(* Logix 5000 project; controller Sucrose_Main Emulate 5570 rev 20.12; software revision 20.01; part 9 of 30 *)
(* tags used below, declared in another part *)
   Alarm_ACK_Master_Timer : TIMER;
   DI_E20_0 : ALIAS FOR FLX_E20:0:I;   // Discrete Input EN2T_FLX 192.168.1.20
   DI_E20_1 : ALIAS FOR FLX_E20:1:I;   // Discrete Input EN2T_FLX 192.168.1.20
   DI_E20_2 : ALIAS FOR FLX_E20:2:I;   // Discrete Input EN2T_FLX 192.168.1.20
   DO_E20_3 : ALIAS FOR FLX_E20:3:O;   // Discrete Output EN2T_FLX 192.168.1.20
   DO_E20_4 : ALIAS FOR FLX_E20:4:O;   // Discrete Output EN2T_FLX 192.168.1.20
   DO_E20_5 : ALIAS FOR FLX_E20:5:O;   // Discrete Output EN2T_FLX 192.168.1.20
   FV230222_AOI : QSI_Flow_Valve;   // FV-23-02-22-O SUCROSE TANK #2 TO TRANSFER PUMP #2 MIX PROOF VALVE OPEN
   FV230412_AOI : QSI_Flow_Valve;   // FV-23-04-12-O SUCROSE TANK #2 TO TRANSFER PUMP #1 MIX PROOF VALVE OPEN
   FV230413_AOI : QSI_Flow_Valve;   // FV-23-04-13-O SUCROSE TANK #3 TO TRANSFER PUMP #1 MIX PROOF VALVE OPEN
   FV230421_AOI : QSI_Flow_Valve;   // FV-23-04-21-O SUCROSE TANK #1 TO TRANSFER PUMP #2 MIX PROOF VALVE OPEN
   FV230423_AOI : QSI_Flow_Valve;   // FV-23-04-23-O SUCROSE TANK #3 TO TRANSFER PUMP #2 MIX PROOF VALVE OPEN
   FV230441_AOI : QSI_Flow_Valve;   // FV-23-04-41-O SUCROSE TRANSFER PUMP #1 DISCHARGE TO FILTRATRION MIX PROOF VALVE OPEN
   FV230442_AOI : QSI_Flow_Valve;   // FV-23-04-42-O SUCROSE TRANSFER PUMP #2 DISCHARGE TO FILTRATRION MIX PROOF VALVE OPEN
   PBL1604001_AOI : QSI_Discrete_Device;   // PBL-16040-01 RESET PB LIGHT
   Sucrose_MM_Enable : BOOL;
   SucroseCIP_P230401_REMOTE : CIP_REMOTE;
   SucroseCIP_P230402_REMOTE : CIP_REMOTE;
   SucroseCIP_RINGMAIN_REMOTE : CIP_REMOTE;
   SucroseDischarge : Area_Program;
   SucroseFiltration : Area_Program;
   SucroseTanks : Area_Program;
(* DischargeArea_EN2T_IO_Discrete_DO_E20_3, continued *)

ROUTINE _03_FV230412   (* ladder *)
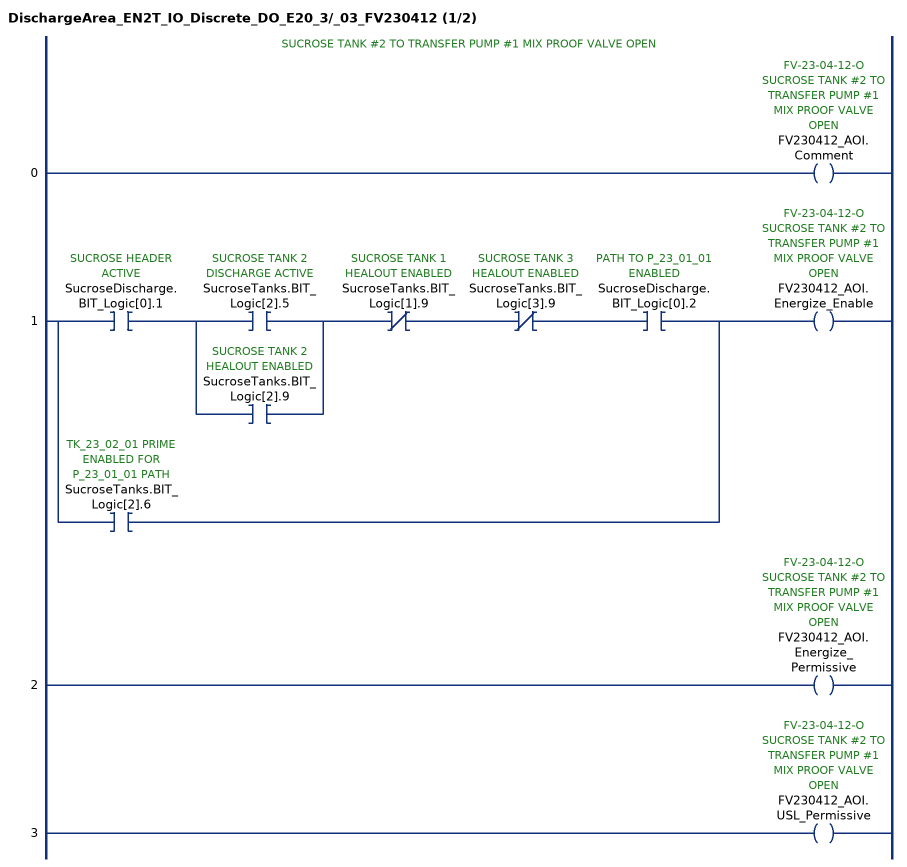
   // SUCROSE TANK #2 TO TRANSFER PUMP #1 MIX PROOF VALVE OPEN
   0: OTE(FV230412_AOI.Comment);
   1: [XIC(SucroseDischarge.BIT_Logic[0].1) [XIC(SucroseTanks.BIT_Logic[2].5) ,XIC(SucroseTanks.BIT_Logic[2].9) ] XIO(SucroseTanks.BIT_Logic[1].9) XIO(SucroseTanks.BIT_Logic[3].9) XIC(SucroseDischarge.BIT_Logic[0].2) ,XIC(SucroseTanks.BIT_Logic[2].6) ]OTE(FV230412_AOI.Energize_Enable);
   2: OTE(FV230412_AOI.Energize_Permissive);
   3: OTE(FV230412_AOI.USL_Permissive);
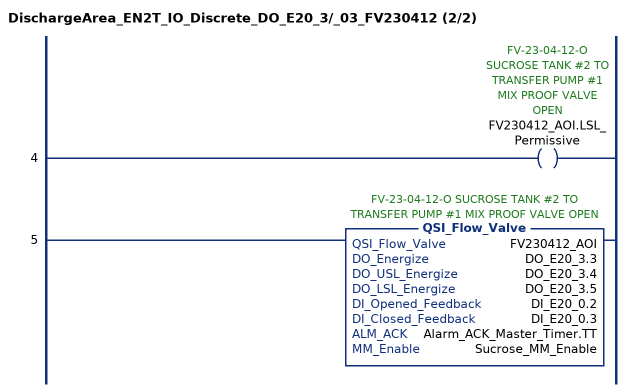
   4: OTE(FV230412_AOI.LSL_Permissive);
   5: QSI_Flow_Valve(FV230412_AOI,DO_E20_3.3,DO_E20_3.4,DO_E20_3.5,DI_E20_0.2,DI_E20_0.3,Alarm_ACK_Master_Timer.TT,Sucrose_MM_Enable);
END_ROUTINE

ROUTINE _06_FV230413   (* ladder *)
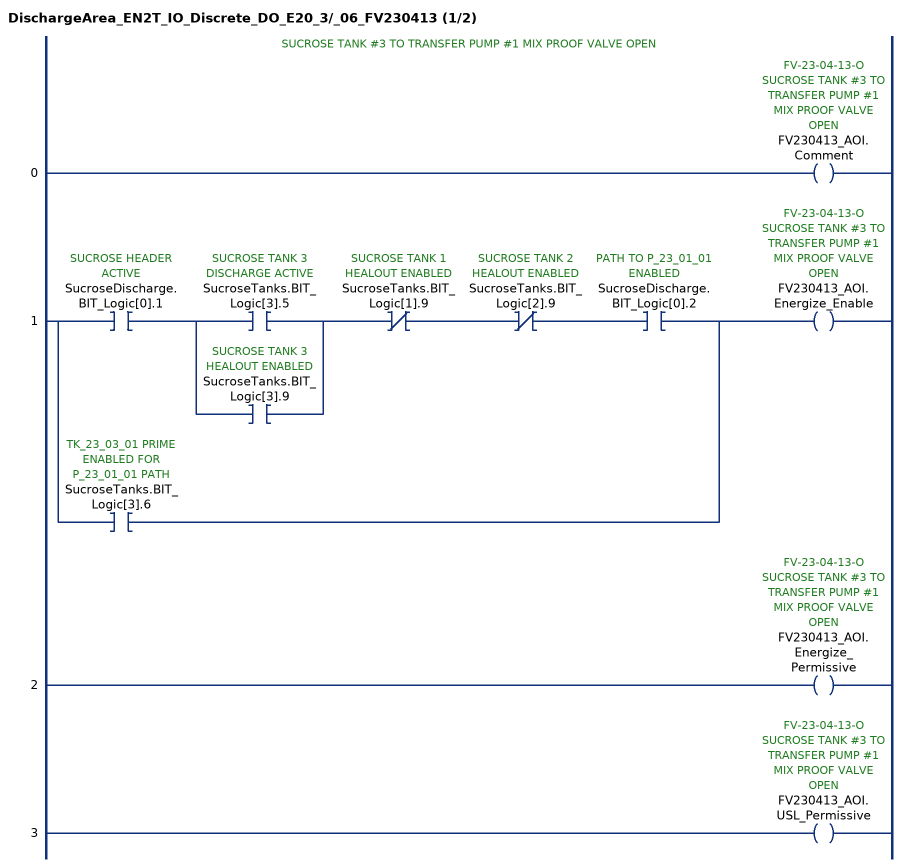
   // SUCROSE TANK #3 TO TRANSFER PUMP #1 MIX PROOF VALVE OPEN
   0: OTE(FV230413_AOI.Comment);
   1: [XIC(SucroseDischarge.BIT_Logic[0].1) [XIC(SucroseTanks.BIT_Logic[3].5) ,XIC(SucroseTanks.BIT_Logic[3].9) ] XIO(SucroseTanks.BIT_Logic[1].9) XIO(SucroseTanks.BIT_Logic[2].9) XIC(SucroseDischarge.BIT_Logic[0].2) ,XIC(SucroseTanks.BIT_Logic[3].6) ]OTE(FV230413_AOI.Energize_Enable);
   2: OTE(FV230413_AOI.Energize_Permissive);
   3: OTE(FV230413_AOI.USL_Permissive);
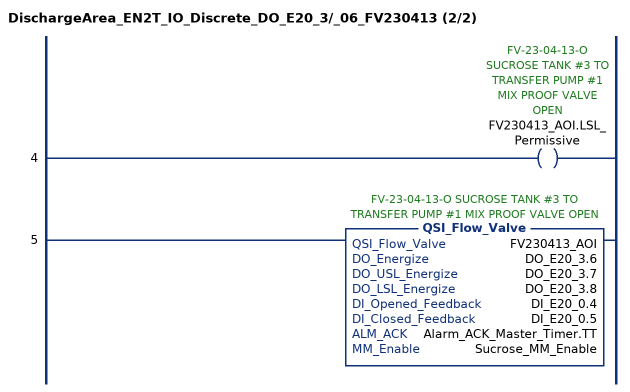
   4: OTE(FV230413_AOI.LSL_Permissive);
   5: QSI_Flow_Valve(FV230413_AOI,DO_E20_3.6,DO_E20_3.7,DO_E20_3.8,DI_E20_0.4,DI_E20_0.5,Alarm_ACK_Master_Timer.TT,Sucrose_MM_Enable);
END_ROUTINE

ROUTINE _09_FV230441   (* ladder *)
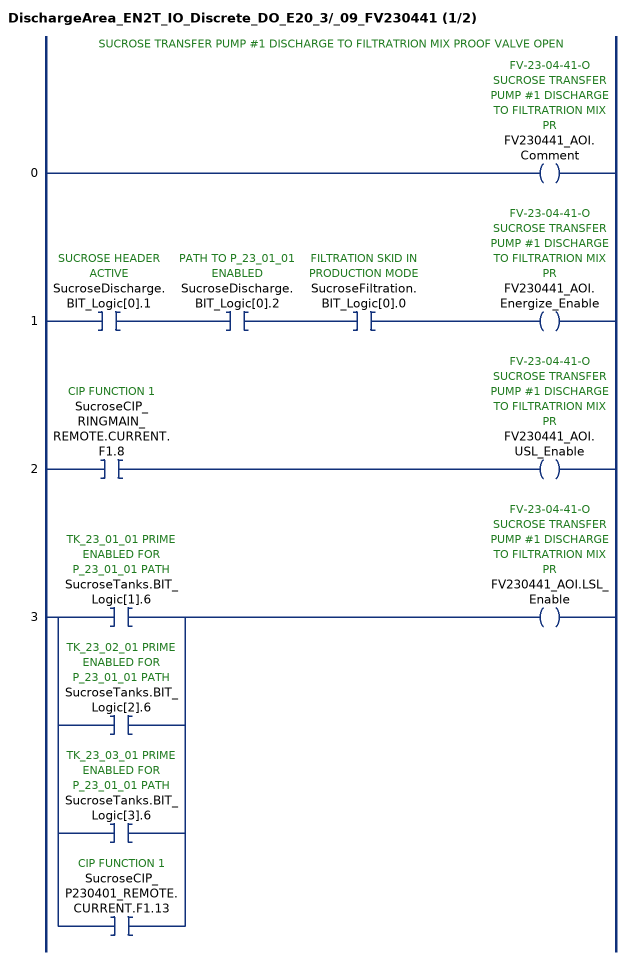
   // SUCROSE TRANSFER PUMP #1 DISCHARGE TO FILTRATRION MIX PROOF VALVE OPEN
   0: OTE(FV230441_AOI.Comment);
   1: XIC(SucroseDischarge.BIT_Logic[0].1)XIC(SucroseDischarge.BIT_Logic[0].2)XIC(SucroseFiltration.BIT_Logic[0].0)OTE(FV230441_AOI.Energize_Enable);
   2: XIC(SucroseCIP_RINGMAIN_REMOTE.CURRENT.F1.8)OTE(FV230441_AOI.USL_Enable);
   3: [XIC(SucroseTanks.BIT_Logic[1].6) ,XIC(SucroseTanks.BIT_Logic[2].6) ,XIC(SucroseTanks.BIT_Logic[3].6) ,XIC(SucroseCIP_P230401_REMOTE.CURRENT.F1.13) ]OTE(FV230441_AOI.LSL_Enable);
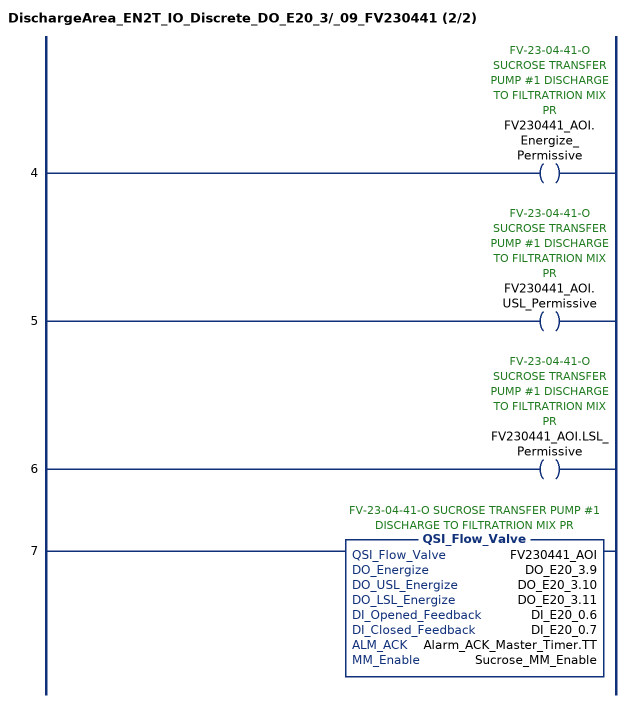
   4: OTE(FV230441_AOI.Energize_Permissive);
   5: OTE(FV230441_AOI.USL_Permissive);
   6: OTE(FV230441_AOI.LSL_Permissive);
   7: QSI_Flow_Valve(FV230441_AOI,DO_E20_3.9,DO_E20_3.10,DO_E20_3.11,DI_E20_0.6,DI_E20_0.7,Alarm_ACK_Master_Timer.TT,Sucrose_MM_Enable);
END_ROUTINE

ROUTINE _12_FV230442   (* ladder *)
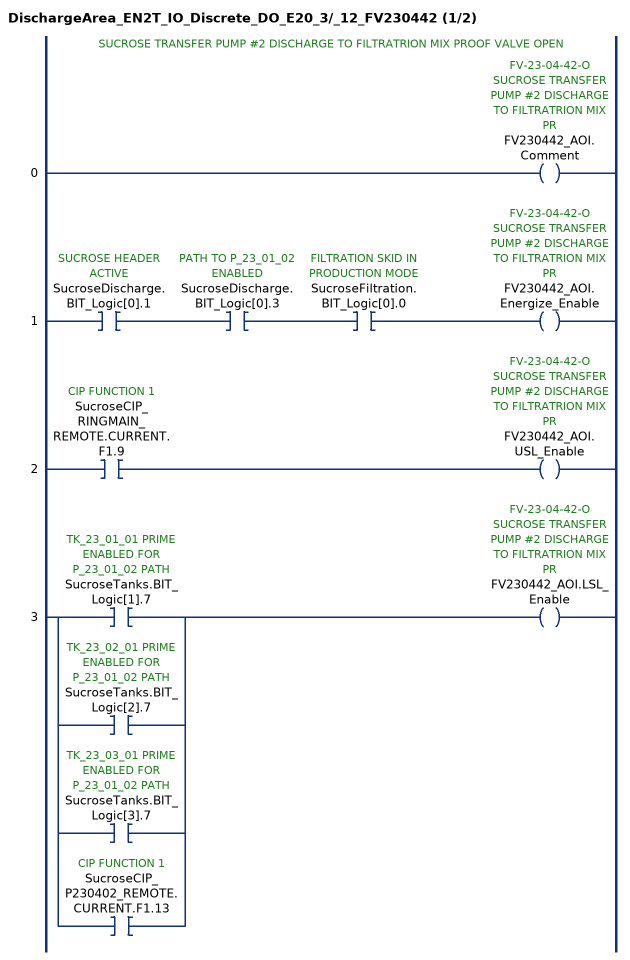
   // SUCROSE TRANSFER PUMP #2 DISCHARGE TO FILTRATRION MIX PROOF VALVE OPEN
   0: OTE(FV230442_AOI.Comment);
   1: XIC(SucroseDischarge.BIT_Logic[0].1)XIC(SucroseDischarge.BIT_Logic[0].3)XIC(SucroseFiltration.BIT_Logic[0].0)OTE(FV230442_AOI.Energize_Enable);
   2: XIC(SucroseCIP_RINGMAIN_REMOTE.CURRENT.F1.9)OTE(FV230442_AOI.USL_Enable);
   3: [XIC(SucroseTanks.BIT_Logic[1].7) ,XIC(SucroseTanks.BIT_Logic[2].7) ,XIC(SucroseTanks.BIT_Logic[3].7) ,XIC(SucroseCIP_P230402_REMOTE.CURRENT.F1.13) ]OTE(FV230442_AOI.LSL_Enable);
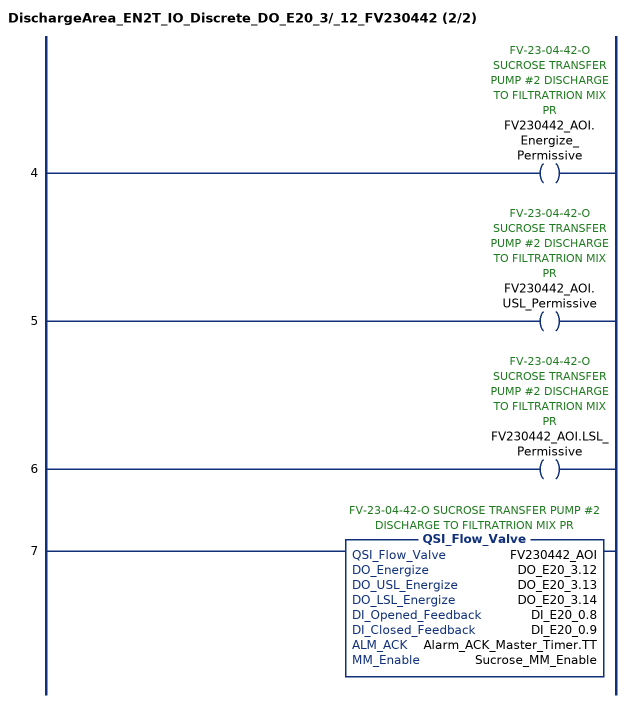
   4: OTE(FV230442_AOI.Energize_Permissive);
   5: OTE(FV230442_AOI.USL_Permissive);
   6: OTE(FV230442_AOI.LSL_Permissive);
   7: QSI_Flow_Valve(FV230442_AOI,DO_E20_3.12,DO_E20_3.13,DO_E20_3.14,DI_E20_0.8,DI_E20_0.9,Alarm_ACK_Master_Timer.TT,Sucrose_MM_Enable);
END_ROUTINE

ROUTINE MainRoutine   (* ladder *)
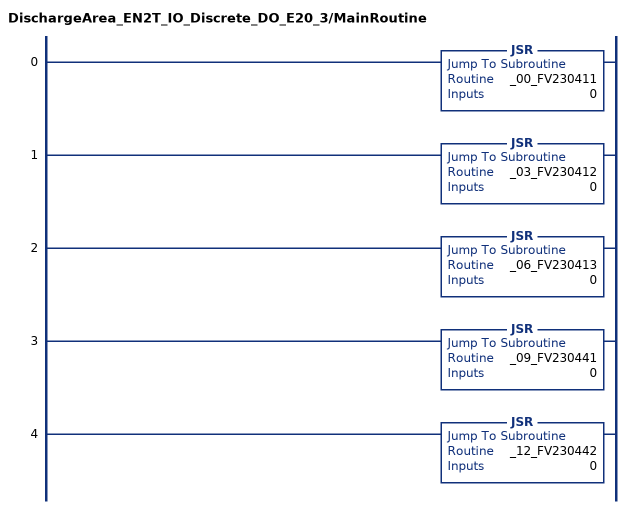
   0: JSR(_00_FV230411,0);
   1: JSR(_03_FV230412,0);
   2: JSR(_06_FV230413,0);
   3: JSR(_09_FV230441,0);
   4: JSR(_12_FV230442,0);
END_ROUTINE
END_PROGRAM

PROGRAM DischargeArea_EN2T_IO_Discrete_DO_E20_4   (* main routine MainRoutine *)

ROUTINE _03_FV230421   (* ladder *)
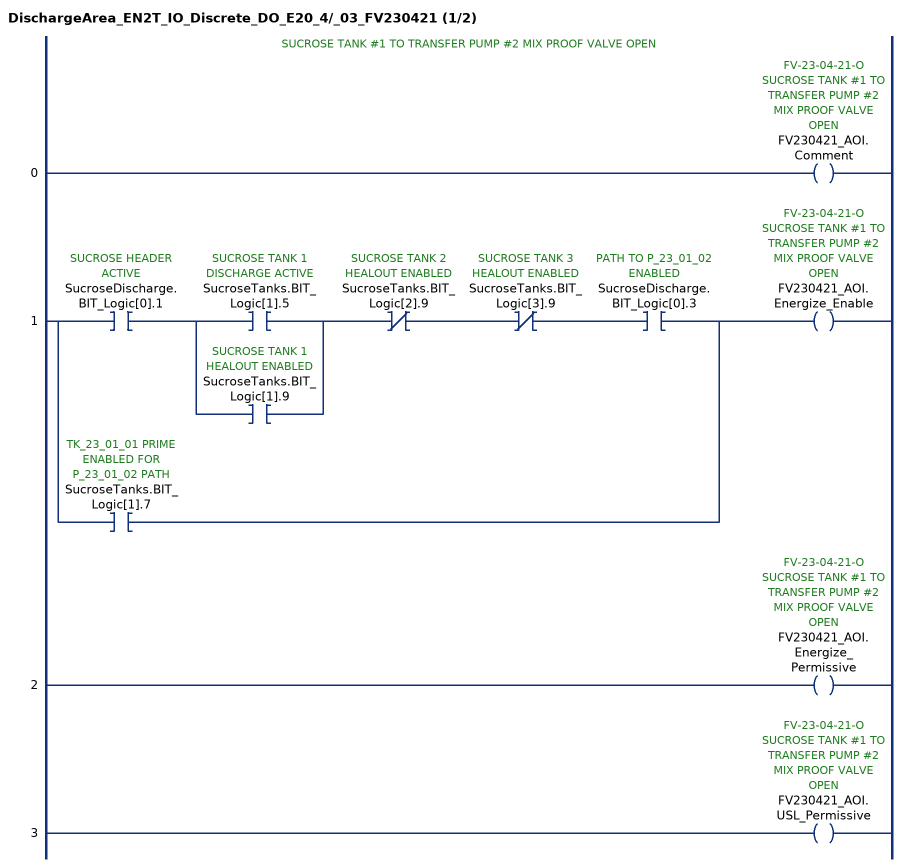
   // SUCROSE TANK #1 TO TRANSFER PUMP #2 MIX PROOF VALVE OPEN
   0: OTE(FV230421_AOI.Comment);
   1: [XIC(SucroseDischarge.BIT_Logic[0].1) [XIC(SucroseTanks.BIT_Logic[1].5) ,XIC(SucroseTanks.BIT_Logic[1].9) ] XIO(SucroseTanks.BIT_Logic[2].9) XIO(SucroseTanks.BIT_Logic[3].9) XIC(SucroseDischarge.BIT_Logic[0].3) ,XIC(SucroseTanks.BIT_Logic[1].7) ]OTE(FV230421_AOI.Energize_Enable);
   2: OTE(FV230421_AOI.Energize_Permissive);
   3: OTE(FV230421_AOI.USL_Permissive);
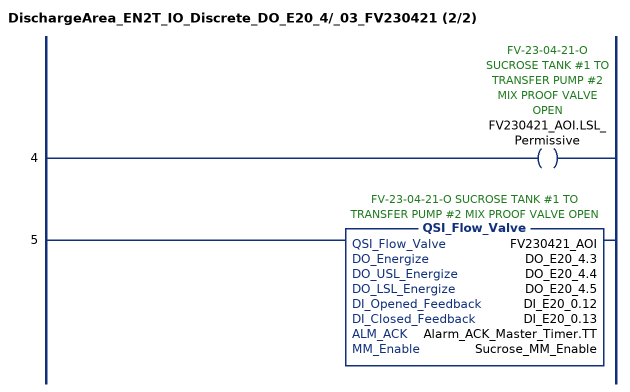
   4: OTE(FV230421_AOI.LSL_Permissive);
   5: QSI_Flow_Valve(FV230421_AOI,DO_E20_4.3,DO_E20_4.4,DO_E20_4.5,DI_E20_0.12,DI_E20_0.13,Alarm_ACK_Master_Timer.TT,Sucrose_MM_Enable);
END_ROUTINE

ROUTINE _06_FV230222   (* ladder *)
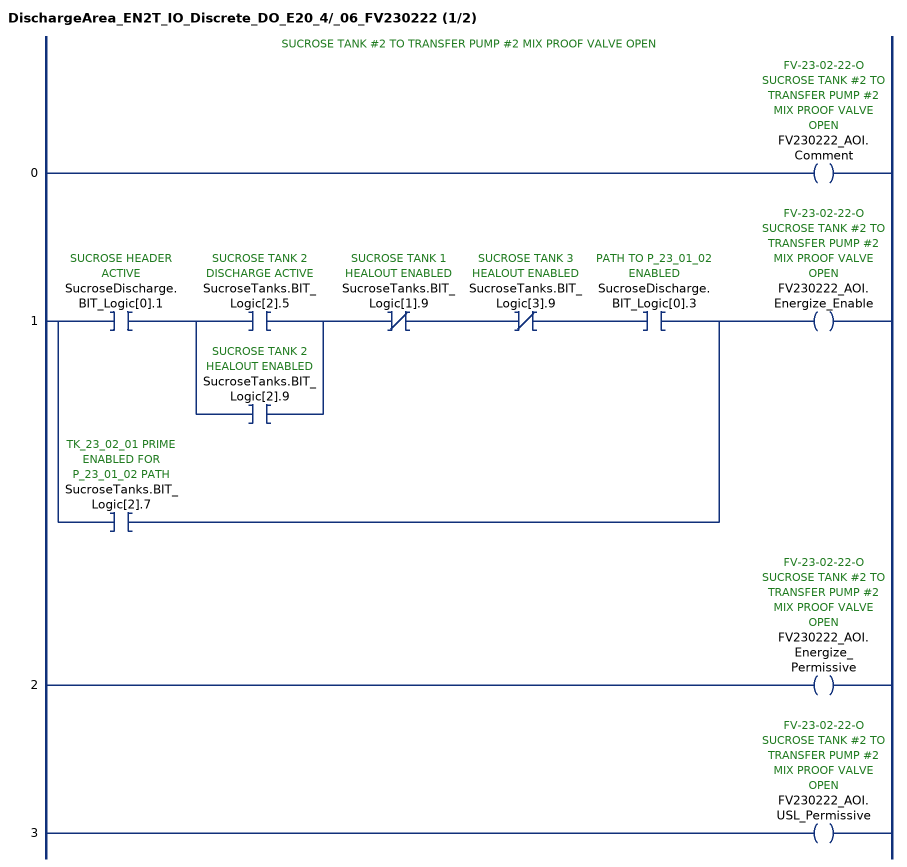
   // SUCROSE TANK #2 TO TRANSFER PUMP #2 MIX PROOF VALVE OPEN
   0: OTE(FV230222_AOI.Comment);
   1: [XIC(SucroseDischarge.BIT_Logic[0].1) [XIC(SucroseTanks.BIT_Logic[2].5) ,XIC(SucroseTanks.BIT_Logic[2].9) ] XIO(SucroseTanks.BIT_Logic[1].9) XIO(SucroseTanks.BIT_Logic[3].9) XIC(SucroseDischarge.BIT_Logic[0].3) ,XIC(SucroseTanks.BIT_Logic[2].7) ]OTE(FV230222_AOI.Energize_Enable);
   2: OTE(FV230222_AOI.Energize_Permissive);
   3: OTE(FV230222_AOI.USL_Permissive);
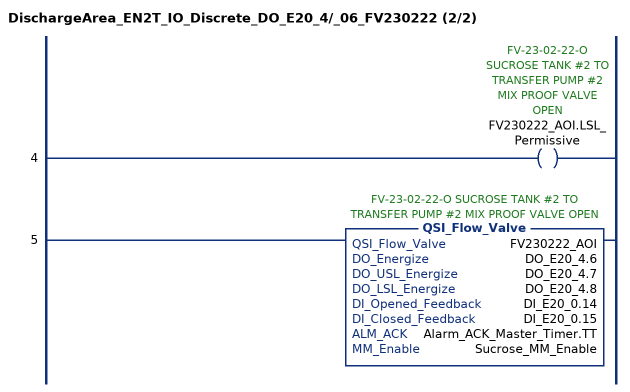
   4: OTE(FV230222_AOI.LSL_Permissive);
   5: QSI_Flow_Valve(FV230222_AOI,DO_E20_4.6,DO_E20_4.7,DO_E20_4.8,DI_E20_0.14,DI_E20_0.15,Alarm_ACK_Master_Timer.TT,Sucrose_MM_Enable);
END_ROUTINE

ROUTINE _09_FV230423   (* ladder *)
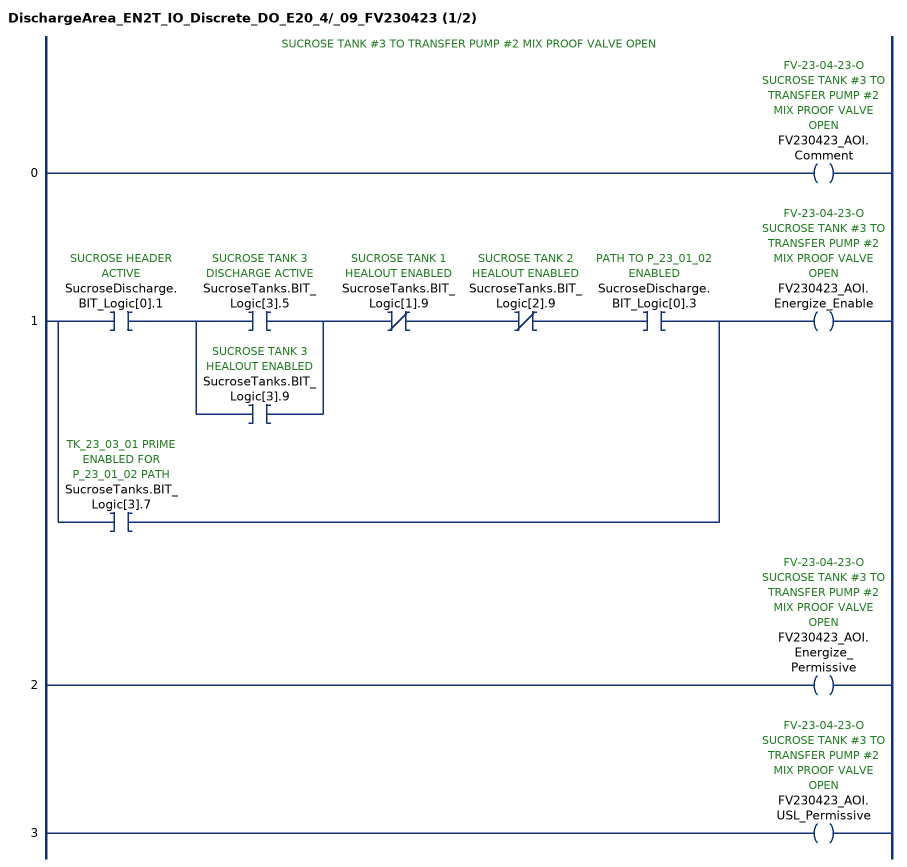
   // SUCROSE TANK #3 TO TRANSFER PUMP #2 MIX PROOF VALVE OPEN
   0: OTE(FV230423_AOI.Comment);
   1: [XIC(SucroseDischarge.BIT_Logic[0].1) [XIC(SucroseTanks.BIT_Logic[3].5) ,XIC(SucroseTanks.BIT_Logic[3].9) ] XIO(SucroseTanks.BIT_Logic[1].9) XIO(SucroseTanks.BIT_Logic[2].9) XIC(SucroseDischarge.BIT_Logic[0].3) ,XIC(SucroseTanks.BIT_Logic[3].7) ]OTE(FV230423_AOI.Energize_Enable);
   2: OTE(FV230423_AOI.Energize_Permissive);
   3: OTE(FV230423_AOI.USL_Permissive);
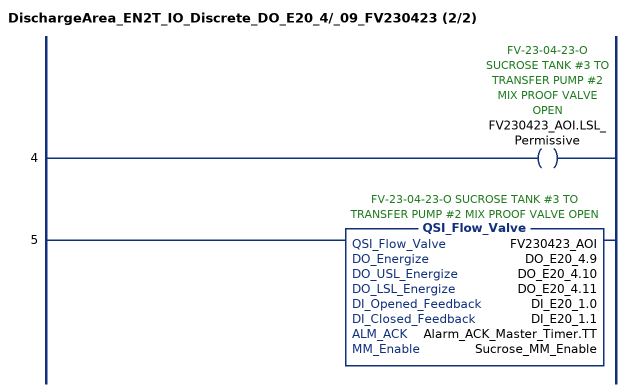
   4: OTE(FV230423_AOI.LSL_Permissive);
   5: QSI_Flow_Valve(FV230423_AOI,DO_E20_4.9,DO_E20_4.10,DO_E20_4.11,DI_E20_1.0,DI_E20_1.1,Alarm_ACK_Master_Timer.TT,Sucrose_MM_Enable);
END_ROUTINE

ROUTINE MainRoutine   (* ladder *)
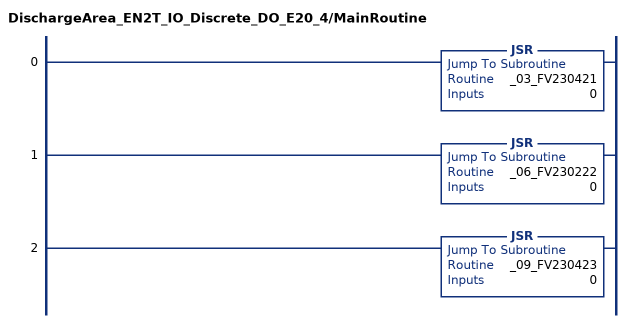
   0: JSR(_03_FV230421,0);
   1: JSR(_06_FV230222,0);
   2: JSR(_09_FV230423,0);
END_ROUTINE
END_PROGRAM

PROGRAM DischargeArea_EN2T_IO_Discrete_DO_E20_5   (* main routine MainRoutine *)

ROUTINE _15_PBL1604001   (* ladder *)
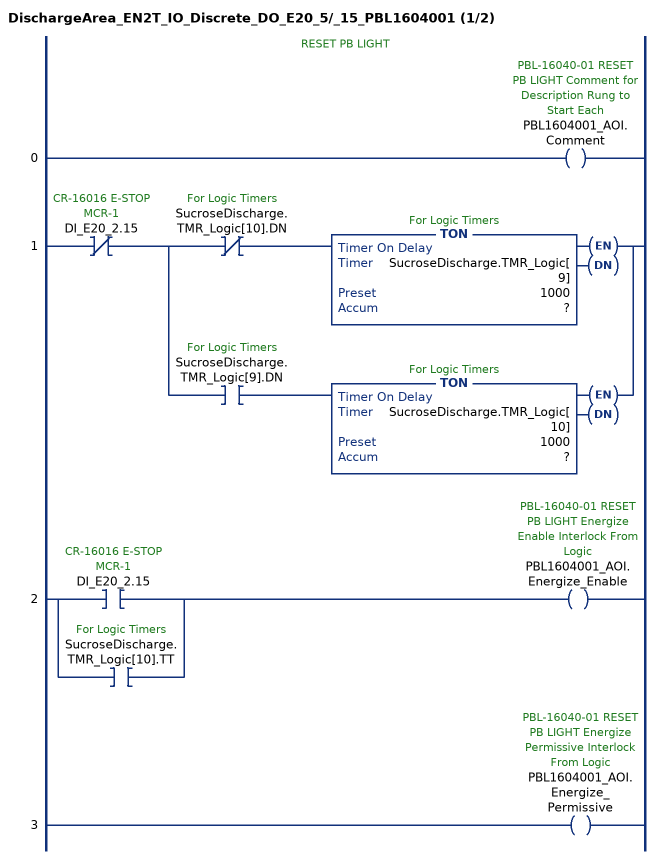
   // RESET PB LIGHT
   0: OTE(PBL1604001_AOI.Comment);
   1: XIO(DI_E20_2.15)[XIO(SucroseDischarge.TMR_Logic[10].DN) TON(SucroseDischarge.TMR_Logic[9],?,?) ,XIC(SucroseDischarge.TMR_Logic[9].DN) TON(SucroseDischarge.TMR_Logic[10],?,?) ];
   2: [XIC(DI_E20_2.15) ,XIC(SucroseDischarge.TMR_Logic[10].TT) ]OTE(PBL1604001_AOI.Energize_Enable);
   3: OTE(PBL1604001_AOI.Energize_Permissive);
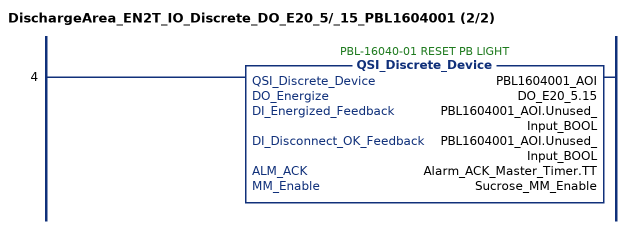
   4: QSI_Discrete_Device(PBL1604001_AOI,DO_E20_5.15,PBL1604001_AOI.Unused_Input_BOOL,PBL1604001_AOI.Unused_Input_BOOL,Alarm_ACK_Master_Timer.TT,Sucrose_MM_Enable);
END_ROUTINE
